GLOBALCONSTANTS wordconst (* Global constants *)
  (* Standard: 61499-1 *)
  (* Version 1.0, 2024-02-22, franz *)
  VAR_GLOBAL CONSTANT
    DWORD_WORD_ZZ : DWORD := 16#0000_0000; (* ZERO Constant *)
    DWORD_WORD_00 : DWORD := 16#0000_FFFF; (* LSB_Byte Constant *)
    DWORD_WORD_01 : DWORD := 16#FFFF_0000; (* MSB_Byte Constant *)
  END_VAR
END_GLOBALCONSTANTS
